Staubli VAL3: GenericApp.dtx

num nDistance
num nDistToDown
num nID = -1
string sConveyorList = "GenericConv"
frame fConveyor = {fatherId=world[0]}
frame fDetection = {fatherId=world[0]}
mdesc mNomSpeed = {blend=off}
mdesc mTracking = {accel=800, vel=800, decel=800, tmax=1000, rmax=500, leave=20, reach=20}
mdesc mTrackOnOff = {leave=20, reach=20}
tool tGripper = {fatherId=flange[0], ioLink=valve1}
